FUNCTION ScaleDP : real
VAR_INPUT
	
END_VAR
VAR
END_VAR

// Raw value of 0 to 32767 scales to -50 to +50

ScaleDP:=

END_FUNCTION

(* stored: Version 1.1.0.1, ProductVersion 3.1.4024.12
   POU ScaleDP: Id {8ae921b4-3b9d-40e3-ac7d-2433d67d89c1}, SpecialFunc None *)
